PROGRAM MAIN
VAR
	nIndex AT %Q*		:	DINT;
	sText AT %Q*		:	T_MaxString;
END_VAR

END_PROGRAM

(* stored: Version 1.1.0.1, ProductVersion 3.1.4024.5
   POU MAIN: Id {2caae984-3533-4153-b882-53095de0599a}, SpecialFunc None *)
